Fanuc KAREL source: userShow.kl

PROGRAM userShow
%NOBUSYLAMP
%NOLOCKGROUP


%from display.klh %import show

BEGIN
	display__show
END userShow
